RoboDK station: Pick_Place_A_Exercicio.rdk

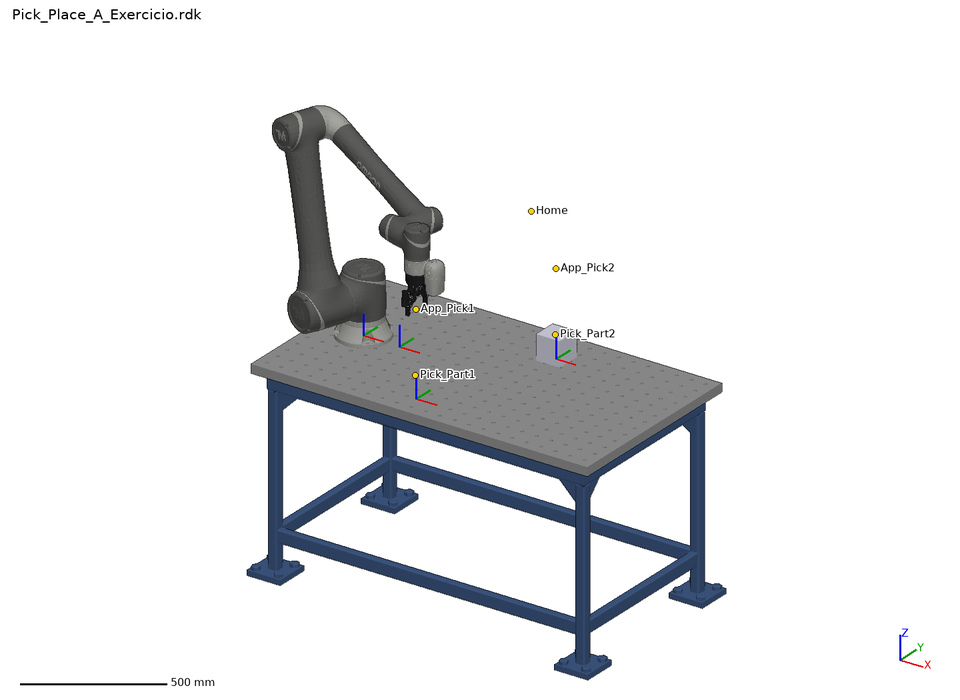
[picture v0: the station drawn from its stored meshes, robots at their saved joint values, targets as dots, program paths as lines]
Station Pick_Place_A_Exercicio (saved by RoboDK 6.0.4). Poses are relative to the parent item; angles as X-Y-Z fixed-axis rotations.
  - frame World at (0, 0, 0) mm
    - object Table 1400x800x800mm at (0, 0, 0) mm, size 1420 x 820 x 800 mm, geometry from Table-1400x800x800mm.sld
    - frame Omron TM12 Base at (-150, 0, 0) mm
      - robot Omron TM12: 6 axes, payload 12 kg, reach 1300 mm, repeatability 0.1 mm, weight 33.3 kg
          modified DH rows (alpha deg, a mm, theta deg, d mm): 0, 0, 0, 165.2; 90, 0, 90, 0; 0, 636.1, 0, 0; 0, 557.9, -90, 156.3; -90, 0, 0, 106; 90, 0, 180, 113.15
          joint limits [-270, -180, -166, -180, -180, -270] to [270, 180, 166, 180, 180, 270]; home [0, 0, 90, -90, 90, 0]; saved at [-17.554, -11.474, 121.737, -19.626, 89.799, -17.553]
        - tool RobotiQ 2F-85 Gripper (Open), TCP at (0, 0, 140) mm, size 147.4 x 75 x 146.8 mm
    - frame Part_1 at (280, -300, 0) mm
      - target App_Pick1 (Cartesian target) at (-0.67, -0.67, 341.07) mm, rotated rx -179.33 ry 0 rz 90 deg; joints [-17.558, -11.106, 122.555, -20.813, 89.799, -17.557] of Omron TM12
      - target Pick_Part1 (Cartesian target) at (-3.6, -0.67, 89.86) mm, rotated rx -179.33 ry 0 rz 90 deg; joints [-17.659, 7.347, 138.541, -55.252, 89.798, -17.658] of Omron TM12
    - target Home (Cartesian target) at (658.05, -156.3, 761.26) mm, rotated rx 175.61 ry 0 rz 90 deg; joints [0, 15.497, 51.569, 18.545, 90, 0] of Omron TM12
    - frame Part_2 at (490, 230, 0) mm
      - target App_Pick2 (Cartesian target) at (-0.67, -0.67, 341.07) mm, rotated rx -179.33 ry 0 rz 90 deg; joints [-17.558, -11.106, 122.555, -20.813, 89.799, -17.557] of Omron TM12
      - target Pick_Part2 (Cartesian target) at (-3.6, -0.67, 89.86) mm, rotated rx -179.33 ry 0 rz 90 deg; joints [-17.659, 7.347, 138.541, -55.252, 89.798, -17.658] of Omron TM12
      - object box at (0, 0, 50) mm, size 100 x 100 x 100 mm, geometry from box.sld
  - program Replace_Object (1 instructions, listed below)
  - program MoveHome (3 instructions, listed below)
  - program Pick (3 instructions, listed below)

--- program Replace_Object (robot Omron TM12) ---
  Replace objects

--- program MoveHome (robot Omron TM12) ---
  Set Ref.: World
  Set Tool: RobotiQ 2F-85 Gripper (Open)
  MoveJ (Home)

--- program Pick (robot Omron TM12) ---
  Set Ref.: Part_1
  Set Tool: RobotiQ 2F-85 Gripper (Open)
  MoveJ (App_Pick1)
